(* IEC 61131-3 sources: AXOpen/src/components.cognex.vision/ctrl/src/AxoVisionPro/TypesStructuresAndEnums, 10 files *)

(* ---- AxoVisionPro_Component_Status.st ---- *)
NAMESPACE AXOpen.Components.Cognex.Vision
    {S7.extern=ReadWrite}
    {#ix-attr:[Container(Layout.Stack)]}
    CLASS PUBLIC AxoVisionPro_Component_Status EXTENDS AXOpen.Components.Abstractions.AxoComponent_Status
        VAR PUBLIC

        END_VAR
    END_CLASS
END_NAMESPACE

(* ---- AxoVisionPro_Config.st ---- *)
NAMESPACE AXOpen.Components.Cognex.Vision
    {S7.extern=ReadWrite}
    {#ix-attr:[Container(Layout.Stack)]}
    CLASS PUBLIC AxoVisionPro_Config
        VAR PUBLIC
            {#ix-set:AttributeName = "<#Info time#>"}
            InfoTime : LTIME := LT#5S;
            {#ix-set:AttributeName = "<#Error time#>"}
            ErrorTime : LTIME := LT#10S;
            {#ix-set:AttributeName = "<#Camera number#>"}
            CameraNo : UINT;
            {#ix-set:AttributeName = "<#Hardware IDs#>"}
            HWIDs : AxoVisionProHWIDs;
        END_VAR
    END_CLASS
END_NAMESPACE

(* ---- AxoVisionPro_Control.st ---- *)
NAMESPACE AXOpen.Components.Cognex.Vision
    {S7.extern=ReadWrite}
    {#ix-attr:[Container(Layout.Stack)]}
    CLASS PUBLIC AxoVisionPro_Control
        VAR PUBLIC
            SoftEvent               : AxoVisionProSoftEventControl;
            SetUserdata             : BOOL;
            InitiateJobLoad         : BOOL;
            InspectionResultsAck    : BOOL;
            ID_Inspection           : BYTE;
            JobLoadID               : WORD;
            WriteDataID             : BYTE;
        END_VAR
    END_CLASS
END_NAMESPACE

(* ---- AxoVisionPro_In.st ---- *)
NAMESPACE AXOpen.Components.Cognex.Vision
    {S7.extern=ReadWrite}
    {#ix-attr:[Container(Layout.Wrap)]}
    CLASS PUBLIC AxoVisionPro_In
        VAR PUBLIC
            {#ix-set:AttributeName = "<#Status#>"}
            {#ix-attr:[ReadOnly()]}
            Status           :   AxoVisionPro_Status;
        END_VAR
    END_CLASS
END_NAMESPACE

(* ---- AxoVisionPro_Out.st ---- *)
NAMESPACE AXOpen.Components.Cognex.Vision
    {S7.extern=ReadWrite}
    {#ix-attr:[Container(Layout.Wrap)]}
    CLASS PUBLIC AxoVisionPro_Out
        VAR PUBLIC
            {#ix-set:AttributeName = "<#Control#>"}
            {#ix-attr:[ReadOnly()]}
            Control           :   AxoVisionPro_Control;
        END_VAR
    END_CLASS
END_NAMESPACE

(* ---- AxoVisionPro_ResultData.st ---- *)
NAMESPACE AXOpen.Components.Cognex.Vision
    {S7.extern=ReadWrite}
    CLASS PUBLIC AxoVisionPro_ResultData EXTENDS AXOpen.Core.AxoByteArray
        VAR PUBLIC
            Data : ARRAY [0..245] OF BYTE;
        END_VAR
    END_CLASS
END_NAMESPACE

(* ---- AxoVisionPro_Status.st ---- *)
NAMESPACE AXOpen.Components.Cognex.Vision
    {S7.extern=ReadWrite}
    {#ix-attr:[Container(Layout.Stack)]}
    CLASS PUBLIC AxoVisionPro_Status
        VAR PUBLIC
            SoftEvent                  : AxoVisionProSoftEventStatus;
            SetUserDataAck             : BOOL;
            Online                     : BOOL;
            SystemBusy                 : BOOL;
            SystemReady                : BOOL;
            JobLoadComplete            : BOOL;
            InspectionOnline           : BOOL;   // Error ID bit z errorID int premennej
            ResultValid                : BOOL;
            ID_Inspection              : WORD;   // rezerva CurentJobID, mozno na kontrolu.
            CurentJobID                : WORD;
            UserDataJobID              : WORD;
            ReadedDataVariantSize      : WORD;   // velkost VARIANT dat ktore chceme vycitat
            WrittenDataVariantSize     : WORD;   // velkost VARIANT dat ktore chceme vycitat
            UserDataLockerJobID        : WORD;   // camera*10 + job
            UserDataLockerIdOperation  : BYTE;
            ReadDataLockerJobID        : WORD;   // camera*10 + job

        END_VAR
    END_CLASS
END_NAMESPACE

(* ---- AxoVisionProHWIDs.st ---- *)
NAMESPACE AXOpen.Components.Cognex.Vision
   {S7.extern=ReadWrite}
	CLASS AxoVisionProHWIDs
      VAR PUBLIC
         {#ix-set:AttributeName = "<#Hardware ID of the device#>"}
         HW_Device              : UINT;
         {#ix-set:AttributeName = "<#Hardware ID 'SystemControl' submodule#>"}
         HW_SystemControl     : UINT;
         {#ix-set:AttributeName = "<#Hardware ID 'EngineControl_1' submodule#>"}
         HW_EngineControl_1   : UINT;
         {#ix-set:AttributeName = "<#Hardware ID 'EngineControl_2' submodule#>"}
         HW_EngineControl_2   : UINT;
         {#ix-set:AttributeName = "<#Hardware ID 'EngineControl_3' submodule#>"}
         HW_EngineControl_3   : UINT;
         {#ix-set:AttributeName = "<#Hardware ID 'EngineControl_4' submodule#>"}
         HW_EngineControl_4   : UINT;
         {#ix-set:AttributeName = "<#Hardware ID 'UserData_240B_1' submodule#>"}
         HW_UserData_240B_1   : UINT;
         {#ix-set:AttributeName = "<#Hardware ID 'UserData_240B_2' submodule#>"}
         HW_UserData_240B_2   : UINT;
         {#ix-set:AttributeName = "<#Hardware ID 'UserData_240B_3' submodule#>"}
         HW_UserData_240B_3   : UINT;
         {#ix-set:AttributeName = "<#Hardware ID 'UserData_240B_4' submodule#>"}
         HW_UserData_240B_4   : UINT;
         {#ix-set:AttributeName = "<#Hardware ID 'UserData_240B_5' submodule#>"}
         HW_UserData_240B_5   : UINT;
         {#ix-set:AttributeName = "<#Hardware ID 'UserData_64B_1' submodule#>"}
         HW_UserData_64B_1    : UINT;
         {#ix-set:AttributeName = "<#Hardware ID 'Results_240B_1' submodule#>"}
         HW_Results_240B_1    : UINT;
         {#ix-set:AttributeName = "<#Hardware ID 'Results_240B_2' submodule#>"}
         HW_Results_240B_2    : UINT;
         {#ix-set:AttributeName = "<#Hardware ID 'Results_240B_3' submodule#>"}
         HW_Results_240B_3    : UINT;
         {#ix-set:AttributeName = "<#Hardware ID 'Results_240B_4' submodule#>"}
         HW_Results_240B_4    : UINT;
         {#ix-set:AttributeName = "<#Hardware ID 'Results_240B_5' submodule#>"}
         HW_Results_240B_5    : UINT;
         {#ix-set:AttributeName = "<#Hardware ID 'Results_64B_1' submodule#>"}
         HW_Results_64B_1     : UINT;
      END_VAR
   END_CLASS
END_NAMESPACE

(* ---- AxoVisionProSoftEventControl.st ---- *)
NAMESPACE AXOpen.Components.Cognex.Vision
   {S7.extern=ReadWrite}
	CLASS AxoVisionProSoftEventControl
      VAR PUBLIC
         Reset          : BOOL;
         DataHandlerAck : BOOL;
         Trigger        : BOOL;
         Reserve        : BOOL;
      END_VAR
   END_CLASS
END_NAMESPACE

(* ---- AxoVisionProSoftEventStatus.st ---- *)
NAMESPACE AXOpen.Components.Cognex.Vision
	CLASS AxoVisionProSoftEventStatus
      VAR PUBLIC
         ResetAck          : BOOL;
         DataHandlerDone   : BOOL;
         TriggerAck        : BOOL;
         Reserve           : BOOL;
      END_VAR
   END_CLASS
END_NAMESPACE
